PROGRAM Recipe1
VAR
	State: INT := 0;
END_VAR

IF IO.Initialized AND NOT IO.Switch THEN
	
	// ponovno zazeni ob tipki...
	// delay...
	// vrni se v stanje ob preklopu...
	// malo spusti, primi, dvigni potem ko ga prime...
	
	// WOOD:
	IF State = 0 THEN
		IF Automatic.ExtensionPositionAuto < 388 THEN
			IO.MotorExtensionDirection := 0;
			IO.MotorExtension := 1;
			Automatic.ExtensionPositionAuto := Automatic.ExtensionPositionAuto + 1;
			Automatic.ExtensionPositionCurrent := Automatic.ExtensionPositionCurrent + 1;
		ELSE
			State := 1;
			IO.MotorExtension := 0;
		END_IF
	ELSIF State = 1 THEN
		IF Automatic.GripPositionAuto < 160 THEN
			IO.MotorGripDirection := 0;
			IO.MotorGrip := 1;
			Automatic.GripPositionAuto := Automatic.GripPositionAuto + 1;
			Automatic.GripPositionCurrent := Automatic.GripPositionCurrent + 1;
		ELSE
			State := 2;
			IO.MotorGripDirection := 1;
			IO.MotorGrip := 0;
		END_IF
	ELSIF State = 2 THEN
		IF NOT IO.EndLiftingSensor THEN
			IO.MotorLiftingDirection := 0;
			IO.MotorLifting := 1;
			Automatic.LiftingPositionAuto := Automatic.LiftingPositionAuto - 1;
			Automatic.LiftingPositionCurrent := Automatic.LiftingPositionCurrent - 1;
		ELSE
			State := 3;
			IO.MotorRotationDirection := 1;
			IO.MotorRotation := 0;
		END_IF
	ELSIF State = 3 THEN
		IF Automatic.RotationPositionAuto < 300 THEN
			IO.MotorRotationDirection := 0;
			IO.MotorRotation := 1;
			Automatic.RotationPositionAuto := Automatic.RotationPositionAuto + 1;
			Automatic.RotationPositionCurrent := Automatic.RotationPositionCurrent + 1;
		ELSE
			State := 4;
			IO.MotorRotationDirection := 1;
			IO.MotorRotation := 0;
		END_IF
	ELSIF State = 4 THEN
		IF NOT IO.EndExtensionSensor THEN
			IO.MotorExtensionDirection := 1;
			IO.MotorExtension := 1;
			Automatic.ExtensionPositionAuto := Automatic.ExtensionPositionAuto - 1;
			Automatic.ExtensionPositionCurrent := Automatic.ExtensionPositionCurrent - 1;
		ELSE
			State := 5;
			IO.MotorExtensionDirection := 0;
			IO.MotorExtension := 0;
		END_IF
	ELSIF State = 5 THEN
		IF NOT IO.EndGripSensor THEN
			IO.MotorGripDirection := 1;
			IO.MotorGrip := 1;
			Automatic.GripPositionAuto := Automatic.GripPositionAuto - 1;
			Automatic.GripPositionCurrent := Automatic.GripPositionCurrent - 1;
		ELSE
			State := 6;
			IO.MotorRotationDirection := 0;
			IO.MotorRotation := 0;
		END_IF
	ELSIF State = 6 THEN
		IF NOT IO.EndRotationSensor THEN
			IO.MotorRotationDirection := 1;
			IO.MotorRotation := 1;
			Automatic.RotationPositionAuto := Automatic.RotationPositionAuto - 1;
			Automatic.RotationPositionCurrent := Automatic.RotationPositionCurrent - 1;
		ELSE
			State := 7;
			IO.MotorRotationDirection := 0;
			IO.MotorRotation := 0;
		END_IF
	END_IF
	
	// PLASTICS:
	IF State = 7 THEN
		IF Automatic.LiftingPositionAuto < 250 THEN
			IO.MotorLiftingDirection := 0;
			IO.MotorLifting := 1;
			Automatic.LiftingPositionAuto := Automatic.LiftingPositionAuto + 1;
			Automatic.LiftingPositionCurrent := Automatic.LiftingPositionCurrent + 1;
		ELSE
			State := 8;
			IO.MotorExtension := 0;
		END_IF
	ELSIF State = 8 THEN
		IF Automatic.ExtensionPositionAuto < 388 THEN
			IO.MotorExtensionDirection := 0;
			IO.MotorExtension := 1;
			Automatic.ExtensionPositionAuto := Automatic.ExtensionPositionAuto + 1;
			Automatic.ExtensionPositionCurrent := Automatic.ExtensionPositionCurrent + 1;
		ELSE
			State := 9;
			IO.MotorExtension := 0;
		END_IF
	ELSIF State = 9 THEN
		IF Automatic.GripPositionAuto < 160 THEN
			IO.MotorGripDirection := 0;
			IO.MotorGrip := 1;
			Automatic.GripPositionAuto := Automatic.GripPositionAuto + 1;
			Automatic.GripPositionCurrent := Automatic.GripPositionCurrent + 1;
		ELSE
			State := 10;
			IO.MotorGripDirection := 1;
			IO.MotorGrip := 0;
		END_IF
	ELSIF State = 10 THEN
		IF NOT IO.EndLiftingSensor THEN
			IO.MotorLiftingDirection := 1;
			IO.MotorLifting := 1;
			Automatic.LiftingPositionAuto := Automatic.LiftingPositionAuto - 1;
			Automatic.LiftingPositionCurrent := Automatic.LiftingPositionCurrent - 1;
		ELSE
			State := 11;
			IO.MotorRotationDirection := 1;
			IO.MotorRotation := 0;
		END_IF
	ELSIF State = 11 THEN
		IF Automatic.RotationPositionAuto < 300 THEN
			IO.MotorRotationDirection := 0;
			IO.MotorRotation := 1;
			Automatic.RotationPositionAuto := Automatic.RotationPositionAuto + 1;
			Automatic.RotationPositionCurrent := Automatic.RotationPositionCurrent + 1;
		ELSE
			State := 12;
			IO.MotorRotationDirection := 1;
			IO.MotorRotation := 0;
		END_IF
	ELSIF State = 12 THEN
		IF Automatic.ExtensionPositionAuto > 300 THEN
			IO.MotorExtensionDirection := 1;
			IO.MotorExtension := 1;
			Automatic.ExtensionPositionAuto := Automatic.ExtensionPositionAuto - 1;
			Automatic.ExtensionPositionCurrent := Automatic.ExtensionPositionCurrent - 1;
		ELSE
			State := 13;
			IO.MotorExtensionDirection := 0;
			IO.MotorExtension := 0;
		END_IF
	ELSIF State = 13 THEN
		IF NOT IO.EndGripSensor THEN
			IO.MotorGripDirection := 1;
			IO.MotorGrip := 1;
			Automatic.GripPositionAuto := Automatic.GripPositionAuto - 1;
			Automatic.GripPositionCurrent := Automatic.GripPositionCurrent - 1;
		ELSE
			State := 14;
			IO.MotorRotationDirection := 0;
			IO.MotorRotation := 0;
		END_IF
	ELSIF State = 14 THEN
		IF NOT IO.EndRotationSensor THEN
			IO.MotorRotationDirection := 1;
			IO.MotorRotation := 1;
			Automatic.RotationPositionAuto := Automatic.RotationPositionAuto - 1;
			Automatic.RotationPositionCurrent := Automatic.RotationPositionCurrent - 1;
		ELSE
			State := 15;
			IO.MotorRotationDirection := 0;
			IO.MotorRotation := 0;
		END_IF
	END_IF
	
	// METAL:
	IF State = 15 THEN
		IF Automatic.LiftingPositionAuto < 400 THEN
			IO.MotorLiftingDirection := 0;
			IO.MotorLifting := 1;
			Automatic.LiftingPositionAuto := Automatic.LiftingPositionAuto + 1;
			Automatic.LiftingPositionCurrent := Automatic.LiftingPositionCurrent + 1;
		ELSE
			State := 16;
			IO.MotorExtension := 0;
		END_IF
	ELSIF State = 16 THEN
		IF Automatic.ExtensionPositionAuto < 388 THEN
			IO.MotorExtensionDirection := 0;
			IO.MotorExtension := 1;
			Automatic.ExtensionPositionAuto := Automatic.ExtensionPositionAuto + 1;
			Automatic.ExtensionPositionCurrent := Automatic.ExtensionPositionCurrent + 1;
		ELSE
			State := 17;
			IO.MotorExtension := 0;
		END_IF
	ELSIF State = 17 THEN
		IF Automatic.GripPositionAuto < 160 THEN
			IO.MotorGripDirection := 0;
			IO.MotorGrip := 1;
			Automatic.GripPositionAuto := Automatic.GripPositionAuto + 1;
			Automatic.GripPositionCurrent := Automatic.GripPositionCurrent + 1;
		ELSE
			State := 18;
			IO.MotorGripDirection := 1;
			IO.MotorGrip := 0;
		END_IF
	ELSIF State = 18 THEN
		IF NOT IO.EndLiftingSensor THEN
			IO.MotorLiftingDirection := 1;
			IO.MotorLifting := 1;
			Automatic.LiftingPositionAuto := Automatic.LiftingPositionAuto - 1;
			Automatic.LiftingPositionCurrent := Automatic.LiftingPositionCurrent - 1;
		ELSE
			State := 19;
			IO.MotorRotationDirection := 1;
			IO.MotorRotation := 0;
		END_IF
	ELSIF State = 19 THEN
		IF Automatic.RotationPositionAuto < 300 THEN
			IO.MotorRotationDirection := 0;
			IO.MotorRotation := 1;
			Automatic.RotationPositionAuto := Automatic.RotationPositionAuto + 1;
			Automatic.RotationPositionCurrent := Automatic.RotationPositionCurrent + 1;
		ELSE
			State := 20;
			IO.MotorRotationDirection := 1;
			IO.MotorRotation := 0;
		END_IF
	ELSIF State = 20 THEN
		IF Automatic.ExtensionPositionAuto > 500 THEN
			IO.MotorExtensionDirection := 1;
			IO.MotorExtension := 1;
			Automatic.ExtensionPositionAuto := Automatic.ExtensionPositionAuto - 1;
			Automatic.ExtensionPositionCurrent := Automatic.ExtensionPositionCurrent - 1;
		ELSE
			State := 21;
			IO.MotorExtensionDirection := 0;
			IO.MotorExtension := 0;
		END_IF
	ELSIF State = 21 THEN
		IF NOT IO.EndGripSensor THEN
			IO.MotorGripDirection := 1;
			IO.MotorGrip := 1;
			Automatic.GripPositionAuto := Automatic.GripPositionAuto - 1;
			Automatic.GripPositionCurrent := Automatic.GripPositionCurrent - 1;
		ELSE
			State := 22;
			IO.MotorRotationDirection := 0;
			IO.MotorRotation := 0;
		END_IF
	ELSIF State = 22 THEN
		IF NOT IO.EndRotationSensor THEN
			IO.MotorRotationDirection := 1;
			IO.MotorRotation := 1;
			Automatic.RotationPositionAuto := Automatic.RotationPositionAuto - 1;
			Automatic.RotationPositionCurrent := Automatic.RotationPositionCurrent - 1;
		ELSE
			State := 23;
			IO.MotorRotationDirection := 0;
			IO.MotorRotation := 0;
		END_IF
	END_IF
END_IF

END_PROGRAM

(* stored: Version 1.1.0.1, ProductVersion 3.1.4024.13
   POU Recipe1: Id {f8183289-6e8d-4e31-9979-1875ef80169a}, SpecialFunc None *)
